//Det6:=a11*a22*a33*a44*a55*a66 - a11*a22*a33*a44*a56*a65 - a11*a22*a33*a45*a54*a66 + a11*a22*a33*a45*a56*a64 + a11*a22*a33*a46*a54*a65 - a11*a22*a33*a46*a55*a64 - a11*a22*a34*a43*a55*a66 + a11*a22*a34*a43*a56*a65 + a11*a22*a34*a45*a53*a66 - a11*a22*a34*a45*a56*a63 - a11*a22*a34*a46*a53*a65 + a11*a22*a34*a46*a55*a63 + a11*a22*a35*a43*a54*a66 - a11*a22*a35*a43*a56*a64 - a11*a22*a35*a44*a53*a66 + a11*a22*a35*a44*a56*a63 + a11*a22*a35*a46*a53*a64 - a11*a22*a35*a46*a54*a63 - a11*a22*a36*a43*a54*a65 + a11*a22*a36*a43*a55*a64 + a11*a22*a36*a44*a53*a65 - a11*a22*a36*a44*a55*a63 - a11*a22*a36*a45*a53*a64 + a11*a22*a36*a45*a54*a63 - a11*a23*a32*a44*a55*a66 + a11*a23*a32*a44*a56*a65 + a11*a23*a32*a45*a54*a66 - a11*a23*a32*a45*a56*a64 - a11*a23*a32*a46*a54*a65 + a11*a23*a32*a46*a55*a64 + a11*a23*a34*a42*a55*a66 - a11*a23*a34*a42*a56*a65 - a11*a23*a34*a45*a52*a66 + a11*a23*a34*a45*a56*a62 + a11*a23*a34*a46*a52*a65 - a11*a23*a34*a46*a55*a62 - a11*a23*a35*a42*a54*a66 + a11*a23*a35*a42*a56*a64 + a11*a23*a35*a44*a52*a66 - a11*a23*a35*a44*a56*a62 - a11*a23*a35*a46*a52*a64 + a11*a23*a35*a46*a54*a62 + a11*a23*a36*a42*a54*a65 - a11*a23*a36*a42*a55*a64 - a11*a23*a36*a44*a52*a65 + a11*a23*a36*a44*a55*a62 + a11*a23*a36*a45*a52*a64 - a11*a23*a36*a45*a54*a62 + a11*a24*a32*a43*a55*a66 - a11*a24*a32*a43*a56*a65 - a11*a24*a32*a45*a53*a66 + a11*a24*a32*a45*a56*a63 + a11*a24*a32*a46*a53*a65 - a11*a24*a32*a46*a55*a63 - a11*a24*a33*a42*a55*a66 + a11*a24*a33*a42*a56*a65 + a11*a24*a33*a45*a52*a66 - a11*a24*a33*a45*a56*a62 - a11*a24*a33*a46*a52*a65 + a11*a24*a33*a46*a55*a62 + a11*a24*a35*a42*a53*a66 - a11*a24*a35*a42*a56*a63 - a11*a24*a35*a43*a52*a66 + a11*a24*a35*a43*a56*a62 + a11*a24*a35*a46*a52*a63 - a11*a24*a35*a46*a53*a62 - a11*a24*a36*a42*a53*a65 + a11*a24*a36*a42*a55*a63 + a11*a24*a36*a43*a52*a65 - a11*a24*a36*a43*a55*a62 - a11*a24*a36*a45*a52*a63 + a11*a24*a36*a45*a53*a62 - a11*a25*a32*a43*a54*a66 + a11*a25*a32*a43*a56*a64 + a11*a25*a32*a44*a53*a66 - a11*a25*a32*a44*a56*a63 - a11*a25*a32*a46*a53*a64 + a11*a25*a32*a46*a54*a63 + a11*a25*a33*a42*a54*a66 - a11*a25*a33*a42*a56*a64 - a11*a25*a33*a44*a52*a66 + a11*a25*a33*a44*a56*a62 + a11*a25*a33*a46*a52*a64 - a11*a25*a33*a46*a54*a62 - a11*a25*a34*a42*a53*a66 + a11*a25*a34*a42*a56*a63 + a11*a25*a34*a43*a52*a66 - a11*a25*a34*a43*a56*a62 - a11*a25*a34*a46*a52*a63 + a11*a25*a34*a46*a53*a62 + a11*a25*a36*a42*a53*a64 - a11*a25*a36*a42*a54*a63 - a11*a25*a36*a43*a52*a64 + a11*a25*a36*a43*a54*a62 + a11*a25*a36*a44*a52*a63 - a11*a25*a36*a44*a53*a62 + a11*a26*a32*a43*a54*a65 - a11*a26*a32*a43*a55*a64 - a11*a26*a32*a44*a53*a65 + a11*a26*a32*a44*a55*a63 + a11*a26*a32*a45*a53*a64 - a11*a26*a32*a45*a54*a63 - a11*a26*a33*a42*a54*a65 + a11*a26*a33*a42*a55*a64 + a11*a26*a33*a44*a52*a65 - a11*a26*a33*a44*a55*a62 - a11*a26*a33*a45*a52*a64 + a11*a26*a33*a45*a54*a62 + a11*a26*a34*a42*a53*a65 - a11*a26*a34*a42*a55*a63 - a11*a26*a34*a43*a52*a65 + a11*a26*a34*a43*a55*a62 + a11*a26*a34*a45*a52*a63 - a11*a26*a34*a45*a53*a62 - a11*a26*a35*a42*a53*a64 + a11*a26*a35*a42*a54*a63 + a11*a26*a35*a43*a52*a64 - a11*a26*a35*a43*a54*a62 - a11*a26*a35*a44*a52*a63 + a11*a26*a35*a44*a53*a62 - a12*a21*a33*a44*a55*a66 + a12*a21*a33*a44*a56*a65 + a12*a21*a33*a45*a54*a66 - a12*a21*a33*a45*a56*a64 - a12*a21*a33*a46*a54*a65 + a12*a21*a33*a46*a55*a64 + a12*a21*a34*a43*a55*a66 - a12*a21*a34*a43*a56*a65 - a12*a21*a34*a45*a53*a66 + a12*a21*a34*a45*a56*a63 + a12*a21*a34*a46*a53*a65 - a12*a21*a34*a46*a55*a63 - a12*a21*a35*a43*a54*a66 + a12*a21*a35*a43*a56*a64 + a12*a21*a35*a44*a53*a66 - a12*a21*a35*a44*a56*a63 - a12*a21*a35*a46*a53*a64 + a12*a21*a35*a46*a54*a63 + a12*a21*a36*a43*a54*a65 - a12*a21*a36*a43*a55*a64 - a12*a21*a36*a44*a53*a65 + a12*a21*a36*a44*a55*a63 + a12*a21*a36*a45*a53*a64 - a12*a21*a36*a45*a54*a63 + a12*a23*a31*a44*a55*a66 - a12*a23*a31*a44*a56*a65 - a12*a23*a31*a45*a54*a66 + a12*a23*a31*a45*a56*a64 + a12*a23*a31*a46*a54*a65 - a12*a23*a31*a46*a55*a64 - a12*a23*a34*a41*a55*a66 + a12*a23*a34*a41*a56*a65 + a12*a23*a34*a45*a51*a66 - a12*a23*a34*a45*a56*a61 - a12*a23*a34*a46*a51*a65 + a12*a23*a34*a46*a55*a61 + a12*a23*a35*a41*a54*a66 - a12*a23*a35*a41*a56*a64 - a12*a23*a35*a44*a51*a66 + a12*a23*a35*a44*a56*a61 + a12*a23*a35*a46*a51*a64 - a12*a23*a35*a46*a54*a61 - a12*a23*a36*a41*a54*a65 + a12*a23*a36*a41*a55*a64 + a12*a23*a36*a44*a51*a65 - a12*a23*a36*a44*a55*a61 - a12*a23*a36*a45*a51*a64 + a12*a23*a36*a45*a54*a61 - a12*a24*a31*a43*a55*a66 + a12*a24*a31*a43*a56*a65 + a12*a24*a31*a45*a53*a66 - a12*a24*a31*a45*a56*a63 - a12*a24*a31*a46*a53*a65 + a12*a24*a31*a46*a55*a63 + a12*a24*a33*a41*a55*a66 - a12*a24*a33*a41*a56*a65 - a12*a24*a33*a45*a51*a66 + a12*a24*a33*a45*a56*a61 + a12*a24*a33*a46*a51*a65 - a12*a24*a33*a46*a55*a61 - a12*a24*a35*a41*a53*a66 + a12*a24*a35*a41*a56*a63 + a12*a24*a35*a43*a51*a66 - a12*a24*a35*a43*a56*a61 - a12*a24*a35*a46*a51*a63 + a12*a24*a35*a46*a53*a61 + a12*a24*a36*a41*a53*a65 - a12*a24*a36*a41*a55*a63 - a12*a24*a36*a43*a51*a65 + a12*a24*a36*a43*a55*a61 + a12*a24*a36*a45*a51*a63 - a12*a24*a36*a45*a53*a61 + a12*a25*a31*a43*a54*a66 - a12*a25*a31*a43*a56*a64 - a12*a25*a31*a44*a53*a66 + a12*a25*a31*a44*a56*a63 + a12*a25*a31*a46*a53*a64 - a12*a25*a31*a46*a54*a63 - a12*a25*a33*a41*a54*a66 + a12*a25*a33*a41*a56*a64 + a12*a25*a33*a44*a51*a66 - a12*a25*a33*a44*a56*a61 - a12*a25*a33*a46*a51*a64 + a12*a25*a33*a46*a54*a61 + a12*a25*a34*a41*a53*a66 - a12*a25*a34*a41*a56*a63 - a12*a25*a34*a43*a51*a66 + a12*a25*a34*a43*a56*a61 + a12*a25*a34*a46*a51*a63 - a12*a25*a34*a46*a53*a61 - a12*a25*a36*a41*a53*a64 + a12*a25*a36*a41*a54*a63 + a12*a25*a36*a43*a51*a64 - a12*a25*a36*a43*a54*a61 - a12*a25*a36*a44*a51*a63 + a12*a25*a36*a44*a53*a61 - a12*a26*a31*a43*a54*a65 + a12*a26*a31*a43*a55*a64 + a12*a26*a31*a44*a53*a65 - a12*a26*a31*a44*a55*a63 - a12*a26*a31*a45*a53*a64 + a12*a26*a31*a45*a54*a63 + a12*a26*a33*a41*a54*a65 - a12*a26*a33*a41*a55*a64 - a12*a26*a33*a44*a51*a65 + a12*a26*a33*a44*a55*a61 + a12*a26*a33*a45*a51*a64 - a12*a26*a33*a45*a54*a61 - a12*a26*a34*a41*a53*a65 + a12*a26*a34*a41*a55*a63 + a12*a26*a34*a43*a51*a65 - a12*a26*a34*a43*a55*a61 - a12*a26*a34*a45*a51*a63 + a12*a26*a34*a45*a53*a61 + a12*a26*a35*a41*a53*a64 - a12*a26*a35*a41*a54*a63 - a12*a26*a35*a43*a51*a64 + a12*a26*a35*a43*a54*a61 + a12*a26*a35*a44*a51*a63 - a12*a26*a35*a44*a53*a61 + a13*a21*a32*a44*a55*a66 - a13*a21*a32*a44*a56*a65 - a13*a21*a32*a45*a54*a66 + a13*a21*a32*a45*a56*a64 + a13*a21*a32*a46*a54*a65 - a13*a21*a32*a46*a55*a64 - a13*a21*a34*a42*a55*a66 + a13*a21*a34*a42*a56*a65 + a13*a21*a34*a45*a52*a66 - a13*a21*a34*a45*a56*a62 - a13*a21*a34*a46*a52*a65 + a13*a21*a34*a46*a55*a62 + a13*a21*a35*a42*a54*a66 - a13*a21*a35*a42*a56*a64 - a13*a21*a35*a44*a52*a66 + a13*a21*a35*a44*a56*a62 + a13*a21*a35*a46*a52*a64 - a13*a21*a35*a46*a54*a62 - a13*a21*a36*a42*a54*a65 + a13*a21*a36*a42*a55*a64 + a13*a21*a36*a44*a52*a65 - a13*a21*a36*a44*a55*a62 - a13*a21*a36*a45*a52*a64 + a13*a21*a36*a45*a54*a62 - a13*a22*a31*a44*a55*a66 + a13*a22*a31*a44*a56*a65 + a13*a22*a31*a45*a54*a66 - a13*a22*a31*a45*a56*a64 - a13*a22*a31*a46*a54*a65 + a13*a22*a31*a46*a55*a64 + a13*a22*a34*a41*a55*a66 - a13*a22*a34*a41*a56*a65 - a13*a22*a34*a45*a51*a66 + a13*a22*a34*a45*a56*a61 + a13*a22*a34*a46*a51*a65 - a13*a22*a34*a46*a55*a61 - a13*a22*a35*a41*a54*a66 + a13*a22*a35*a41*a56*a64 + a13*a22*a35*a44*a51*a66 - a13*a22*a35*a44*a56*a61 - a13*a22*a35*a46*a51*a64 + a13*a22*a35*a46*a54*a61 + a13*a22*a36*a41*a54*a65 - a13*a22*a36*a41*a55*a64 - a13*a22*a36*a44*a51*a65 + a13*a22*a36*a44*a55*a61 + a13*a22*a36*a45*a51*a64 - a13*a22*a36*a45*a54*a61 + a13*a24*a31*a42*a55*a66 - a13*a24*a31*a42*a56*a65 - a13*a24*a31*a45*a52*a66 + a13*a24*a31*a45*a56*a62 + a13*a24*a31*a46*a52*a65 - a13*a24*a31*a46*a55*a62 - a13*a24*a32*a41*a55*a66 + a13*a24*a32*a41*a56*a65 + a13*a24*a32*a45*a51*a66 - a13*a24*a32*a45*a56*a61 - a13*a24*a32*a46*a51*a65 + a13*a24*a32*a46*a55*a61 + a13*a24*a35*a41*a52*a66 - a13*a24*a35*a41*a56*a62 - a13*a24*a35*a42*a51*a66 + a13*a24*a35*a42*a56*a61 + a13*a24*a35*a46*a51*a62 - a13*a24*a35*a46*a52*a61 - a13*a24*a36*a41*a52*a65 + a13*a24*a36*a41*a55*a62 + a13*a24*a36*a42*a51*a65 - a13*a24*a36*a42*a55*a61 - a13*a24*a36*a45*a51*a62 + a13*a24*a36*a45*a52*a61 - a13*a25*a31*a42*a54*a66 + a13*a25*a31*a42*a56*a64 + a13*a25*a31*a44*a52*a66 - a13*a25*a31*a44*a56*a62 - a13*a25*a31*a46*a52*a64 + a13*a25*a31*a46*a54*a62 + a13*a25*a32*a41*a54*a66 - a13*a25*a32*a41*a56*a64 - a13*a25*a32*a44*a51*a66 + a13*a25*a32*a44*a56*a61 + a13*a25*a32*a46*a51*a64 - a13*a25*a32*a46*a54*a61 - a13*a25*a34*a41*a52*a66 + a13*a25*a34*a41*a56*a62 + a13*a25*a34*a42*a51*a66 - a13*a25*a34*a42*a56*a61 - a13*a25*a34*a46*a51*a62 + a13*a25*a34*a46*a52*a61 + a13*a25*a36*a41*a52*a64 - a13*a25*a36*a41*a54*a62 - a13*a25*a36*a42*a51*a64 + a13*a25*a36*a42*a54*a61 + a13*a25*a36*a44*a51*a62 - a13*a25*a36*a44*a52*a61 + a13*a26*a31*a42*a54*a65 - a13*a26*a31*a42*a55*a64 - a13*a26*a31*a44*a52*a65 + a13*a26*a31*a44*a55*a62 + a13*a26*a31*a45*a52*a64 - a13*a26*a31*a45*a54*a62 - a13*a26*a32*a41*a54*a65 + a13*a26*a32*a41*a55*a64 + a13*a26*a32*a44*a51*a65 - a13*a26*a32*a44*a55*a61 - a13*a26*a32*a45*a51*a64 + a13*a26*a32*a45*a54*a61 + a13*a26*a34*a41*a52*a65 - a13*a26*a34*a41*a55*a62 - a13*a26*a34*a42*a51*a65 + a13*a26*a34*a42*a55*a61 + a13*a26*a34*a45*a51*a62 - a13*a26*a34*a45*a52*a61 - a13*a26*a35*a41*a52*a64 + a13*a26*a35*a41*a54*a62 + a13*a26*a35*a42*a51*a64 - a13*a26*a35*a42*a54*a61 - a13*a26*a35*a44*a51*a62 + a13*a26*a35*a44*a52*a61 - a14*a21*a32*a43*a55*a66 + a14*a21*a32*a43*a56*a65 + a14*a21*a32*a45*a53*a66 - a14*a21*a32*a45*a56*a63 - a14*a21*a32*a46*a53*a65 + a14*a21*a32*a46*a55*a63 + a14*a21*a33*a42*a55*a66 - a14*a21*a33*a42*a56*a65 - a14*a21*a33*a45*a52*a66 + a14*a21*a33*a45*a56*a62 + a14*a21*a33*a46*a52*a65 - a14*a21*a33*a46*a55*a62 - a14*a21*a35*a42*a53*a66 + a14*a21*a35*a42*a56*a63 + a14*a21*a35*a43*a52*a66 - a14*a21*a35*a43*a56*a62 - a14*a21*a35*a46*a52*a63 + a14*a21*a35*a46*a53*a62 + a14*a21*a36*a42*a53*a65 - a14*a21*a36*a42*a55*a63 - a14*a21*a36*a43*a52*a65 + a14*a21*a36*a43*a55*a62 + a14*a21*a36*a45*a52*a63 - a14*a21*a36*a45*a53*a62 + a14*a22*a31*a43*a55*a66 - a14*a22*a31*a43*a56*a65 - a14*a22*a31*a45*a53*a66 + a14*a22*a31*a45*a56*a63 + a14*a22*a31*a46*a53*a65 - a14*a22*a31*a46*a55*a63 - a14*a22*a33*a41*a55*a66 + a14*a22*a33*a41*a56*a65 + a14*a22*a33*a45*a51*a66 - a14*a22*a33*a45*a56*a61 - a14*a22*a33*a46*a51*a65 + a14*a22*a33*a46*a55*a61 + a14*a22*a35*a41*a53*a66 - a14*a22*a35*a41*a56*a63 - a14*a22*a35*a43*a51*a66 + a14*a22*a35*a43*a56*a61 + a14*a22*a35*a46*a51*a63 - a14*a22*a35*a46*a53*a61 - a14*a22*a36*a41*a53*a65 + a14*a22*a36*a41*a55*a63 + a14*a22*a36*a43*a51*a65 - a14*a22*a36*a43*a55*a61 - a14*a22*a36*a45*a51*a63 + a14*a22*a36*a45*a53*a61 - a14*a23*a31*a42*a55*a66 + a14*a23*a31*a42*a56*a65 + a14*a23*a31*a45*a52*a66 - a14*a23*a31*a45*a56*a62 - a14*a23*a31*a46*a52*a65 + a14*a23*a31*a46*a55*a62 + a14*a23*a32*a41*a55*a66 - a14*a23*a32*a41*a56*a65 - a14*a23*a32*a45*a51*a66 + a14*a23*a32*a45*a56*a61 + a14*a23*a32*a46*a51*a65 - a14*a23*a32*a46*a55*a61 - a14*a23*a35*a41*a52*a66 + a14*a23*a35*a41*a56*a62 + a14*a23*a35*a42*a51*a66 - a14*a23*a35*a42*a56*a61 - a14*a23*a35*a46*a51*a62 + a14*a23*a35*a46*a52*a61 + a14*a23*a36*a41*a52*a65 - a14*a23*a36*a41*a55*a62 - a14*a23*a36*a42*a51*a65 + a14*a23*a36*a42*a55*a61 + a14*a23*a36*a45*a51*a62 - a14*a23*a36*a45*a52*a61 + a14*a25*a31*a42*a53*a66 - a14*a25*a31*a42*a56*a63 - a14*a25*a31*a43*a52*a66 + a14*a25*a31*a43*a56*a62 + a14*a25*a31*a46*a52*a63 - a14*a25*a31*a46*a53*a62 - a14*a25*a32*a41*a53*a66 + a14*a25*a32*a41*a56*a63 + a14*a25*a32*a43*a51*a66 - a14*a25*a32*a43*a56*a61 - a14*a25*a32*a46*a51*a63 + a14*a25*a32*a46*a53*a61 + a14*a25*a33*a41*a52*a66 - a14*a25*a33*a41*a56*a62 - a14*a25*a33*a42*a51*a66 + a14*a25*a33*a42*a56*a61 + a14*a25*a33*a46*a51*a62 - a14*a25*a33*a46*a52*a61 - a14*a25*a36*a41*a52*a63 + a14*a25*a36*a41*a53*a62 + a14*a25*a36*a42*a51*a63 - a14*a25*a36*a42*a53*a61 - a14*a25*a36*a43*a51*a62 + a14*a25*a36*a43*a52*a61 - a14*a26*a31*a42*a53*a65 + a14*a26*a31*a42*a55*a63 + a14*a26*a31*a43*a52*a65 - a14*a26*a31*a43*a55*a62 - a14*a26*a31*a45*a52*a63 + a14*a26*a31*a45*a53*a62 + a14*a26*a32*a41*a53*a65 - a14*a26*a32*a41*a55*a63 - a14*a26*a32*a43*a51*a65 + a14*a26*a32*a43*a55*a61 + a14*a26*a32*a45*a51*a63 - a14*a26*a32*a45*a53*a61 - a14*a26*a33*a41*a52*a65 + a14*a26*a33*a41*a55*a62 + a14*a26*a33*a42*a51*a65 - a14*a26*a33*a42*a55*a61 - a14*a26*a33*a45*a51*a62 + a14*a26*a33*a45*a52*a61 + a14*a26*a35*a41*a52*a63 - a14*a26*a35*a41*a53*a62 - a14*a26*a35*a42*a51*a63 + a14*a26*a35*a42*a53*a61 + a14*a26*a35*a43*a51*a62 - a14*a26*a35*a43*a52*a61 + a15*a21*a32*a43*a54*a66 - a15*a21*a32*a43*a56*a64 - a15*a21*a32*a44*a53*a66 + a15*a21*a32*a44*a56*a63 + a15*a21*a32*a46*a53*a64 - a15*a21*a32*a46*a54*a63 - a15*a21*a33*a42*a54*a66 + a15*a21*a33*a42*a56*a64 + a15*a21*a33*a44*a52*a66 - a15*a21*a33*a44*a56*a62 - a15*a21*a33*a46*a52*a64 + a15*a21*a33*a46*a54*a62 + a15*a21*a34*a42*a53*a66 - a15*a21*a34*a42*a56*a63 - a15*a21*a34*a43*a52*a66 + a15*a21*a34*a43*a56*a62 + a15*a21*a34*a46*a52*a63 - a15*a21*a34*a46*a53*a62 - a15*a21*a36*a42*a53*a64 + a15*a21*a36*a42*a54*a63 + a15*a21*a36*a43*a52*a64 - a15*a21*a36*a43*a54*a62 - a15*a21*a36*a44*a52*a63 + a15*a21*a36*a44*a53*a62 - a15*a22*a31*a43*a54*a66 + a15*a22*a31*a43*a56*a64 + a15*a22*a31*a44*a53*a66 - a15*a22*a31*a44*a56*a63 - a15*a22*a31*a46*a53*a64 + a15*a22*a31*a46*a54*a63 + a15*a22*a33*a41*a54*a66 - a15*a22*a33*a41*a56*a64 - a15*a22*a33*a44*a51*a66 + a15*a22*a33*a44*a56*a61 + a15*a22*a33*a46*a51*a64 - a15*a22*a33*a46*a54*a61 - a15*a22*a34*a41*a53*a66 + a15*a22*a34*a41*a56*a63 + a15*a22*a34*a43*a51*a66 - a15*a22*a34*a43*a56*a61 - a15*a22*a34*a46*a51*a63 + a15*a22*a34*a46*a53*a61 + a15*a22*a36*a41*a53*a64 - a15*a22*a36*a41*a54*a63 - a15*a22*a36*a43*a51*a64 + a15*a22*a36*a43*a54*a61 + a15*a22*a36*a44*a51*a63 - a15*a22*a36*a44*a53*a61 + a15*a23*a31*a42*a54*a66 - a15*a23*a31*a42*a56*a64 - a15*a23*a31*a44*a52*a66 + a15*a23*a31*a44*a56*a62 + a15*a23*a31*a46*a52*a64 - a15*a23*a31*a46*a54*a62 - a15*a23*a32*a41*a54*a66 + a15*a23*a32*a41*a56*a64 + a15*a23*a32*a44*a51*a66 - a15*a23*a32*a44*a56*a61 - a15*a23*a32*a46*a51*a64 + a15*a23*a32*a46*a54*a61 + a15*a23*a34*a41*a52*a66 - a15*a23*a34*a41*a56*a62 - a15*a23*a34*a42*a51*a66 + a15*a23*a34*a42*a56*a61 + a15*a23*a34*a46*a51*a62 - a15*a23*a34*a46*a52*a61 - a15*a23*a36*a41*a52*a64 + a15*a23*a36*a41*a54*a62 + a15*a23*a36*a42*a51*a64 - a15*a23*a36*a42*a54*a61 - a15*a23*a36*a44*a51*a62 + a15*a23*a36*a44*a52*a61 - a15*a24*a31*a42*a53*a66 + a15*a24*a31*a42*a56*a63 + a15*a24*a31*a43*a52*a66 - a15*a24*a31*a43*a56*a62 - a15*a24*a31*a46*a52*a63 + a15*a24*a31*a46*a53*a62 + a15*a24*a32*a41*a53*a66 - a15*a24*a32*a41*a56*a63 - a15*a24*a32*a43*a51*a66 + a15*a24*a32*a43*a56*a61 + a15*a24*a32*a46*a51*a63 - a15*a24*a32*a46*a53*a61 - a15*a24*a33*a41*a52*a66 + a15*a24*a33*a41*a56*a62 + a15*a24*a33*a42*a51*a66 - a15*a24*a33*a42*a56*a61 - a15*a24*a33*a46*a51*a62 + a15*a24*a33*a46*a52*a61 + a15*a24*a36*a41*a52*a63 - a15*a24*a36*a41*a53*a62 - a15*a24*a36*a42*a51*a63 + a15*a24*a36*a42*a53*a61 + a15*a24*a36*a43*a51*a62 - a15*a24*a36*a43*a52*a61 + a15*a26*a31*a42*a53*a64 - a15*a26*a31*a42*a54*a63 - a15*a26*a31*a43*a52*a64 + a15*a26*a31*a43*a54*a62 + a15*a26*a31*a44*a52*a63 - a15*a26*a31*a44*a53*a62 - a15*a26*a32*a41*a53*a64 + a15*a26*a32*a41*a54*a63 + a15*a26*a32*a43*a51*a64 - a15*a26*a32*a43*a54*a61 - a15*a26*a32*a44*a51*a63 + a15*a26*a32*a44*a53*a61 + a15*a26*a33*a41*a52*a64 - a15*a26*a33*a41*a54*a62 - a15*a26*a33*a42*a51*a64 + a15*a26*a33*a42*a54*a61 + a15*a26*a33*a44*a51*a62 - a15*a26*a33*a44*a52*a61 - a15*a26*a34*a41*a52*a63 + a15*a26*a34*a41*a53*a62 + a15*a26*a34*a42*a51*a63 - a15*a26*a34*a42*a53*a61 - a15*a26*a34*a43*a51*a62 + a15*a26*a34*a43*a52*a61 - a16*a21*a32*a43*a54*a65 + a16*a21*a32*a43*a55*a64 + a16*a21*a32*a44*a53*a65 - a16*a21*a32*a44*a55*a63 - a16*a21*a32*a45*a53*a64 + a16*a21*a32*a45*a54*a63 + a16*a21*a33*a42*a54*a65 - a16*a21*a33*a42*a55*a64 - a16*a21*a33*a44*a52*a65 + a16*a21*a33*a44*a55*a62 + a16*a21*a33*a45*a52*a64 - a16*a21*a33*a45*a54*a62 - a16*a21*a34*a42*a53*a65 + a16*a21*a34*a42*a55*a63 + a16*a21*a34*a43*a52*a65 - a16*a21*a34*a43*a55*a62 - a16*a21*a34*a45*a52*a63 + a16*a21*a34*a45*a53*a62 + a16*a21*a35*a42*a53*a64 - a16*a21*a35*a42*a54*a63 - a16*a21*a35*a43*a52*a64 + a16*a21*a35*a43*a54*a62 + a16*a21*a35*a44*a52*a63 - a16*a21*a35*a44*a53*a62 + a16*a22*a31*a43*a54*a65 - a16*a22*a31*a43*a55*a64 - a16*a22*a31*a44*a53*a65 + a16*a22*a31*a44*a55*a63 + a16*a22*a31*a45*a53*a64 - a16*a22*a31*a45*a54*a63 - a16*a22*a33*a41*a54*a65 + a16*a22*a33*a41*a55*a64 + a16*a22*a33*a44*a51*a65 - a16*a22*a33*a44*a55*a61 - a16*a22*a33*a45*a51*a64 + a16*a22*a33*a45*a54*a61 + a16*a22*a34*a41*a53*a65 - a16*a22*a34*a41*a55*a63 - a16*a22*a34*a43*a51*a65 + a16*a22*a34*a43*a55*a61 + a16*a22*a34*a45*a51*a63 - a16*a22*a34*a45*a53*a61 - a16*a22*a35*a41*a53*a64 + a16*a22*a35*a41*a54*a63 + a16*a22*a35*a43*a51*a64 - a16*a22*a35*a43*a54*a61 - a16*a22*a35*a44*a51*a63 + a16*a22*a35*a44*a53*a61 - a16*a23*a31*a42*a54*a65 + a16*a23*a31*a42*a55*a64 + a16*a23*a31*a44*a52*a65 - a16*a23*a31*a44*a55*a62 - a16*a23*a31*a45*a52*a64 + a16*a23*a31*a45*a54*a62 + a16*a23*a32*a41*a54*a65 - a16*a23*a32*a41*a55*a64 - a16*a23*a32*a44*a51*a65 + a16*a23*a32*a44*a55*a61 + a16*a23*a32*a45*a51*a64 - a16*a23*a32*a45*a54*a61 - a16*a23*a34*a41*a52*a65 + a16*a23*a34*a41*a55*a62 + a16*a23*a34*a42*a51*a65 - a16*a23*a34*a42*a55*a61 - a16*a23*a34*a45*a51*a62 + a16*a23*a34*a45*a52*a61 + a16*a23*a35*a41*a52*a64 - a16*a23*a35*a41*a54*a62 - a16*a23*a35*a42*a51*a64 + a16*a23*a35*a42*a54*a61 + a16*a23*a35*a44*a51*a62 - a16*a23*a35*a44*a52*a61 + a16*a24*a31*a42*a53*a65 - a16*a24*a31*a42*a55*a63 - a16*a24*a31*a43*a52*a65 + a16*a24*a31*a43*a55*a62 + a16*a24*a31*a45*a52*a63 - a16*a24*a31*a45*a53*a62 - a16*a24*a32*a41*a53*a65 + a16*a24*a32*a41*a55*a63 + a16*a24*a32*a43*a51*a65 - a16*a24*a32*a43*a55*a61 - a16*a24*a32*a45*a51*a63 + a16*a24*a32*a45*a53*a61 + a16*a24*a33*a41*a52*a65 - a16*a24*a33*a41*a55*a62 - a16*a24*a33*a42*a51*a65 + a16*a24*a33*a42*a55*a61 + a16*a24*a33*a45*a51*a62 - a16*a24*a33*a45*a52*a61 - a16*a24*a35*a41*a52*a63 + a16*a24*a35*a41*a53*a62 + a16*a24*a35*a42*a51*a63 - a16*a24*a35*a42*a53*a61 - a16*a24*a35*a43*a51*a62 + a16*a24*a35*a43*a52*a61 - a16*a25*a31*a42*a53*a64 + a16*a25*a31*a42*a54*a63 + a16*a25*a31*a43*a52*a64 - a16*a25*a31*a43*a54*a62 - a16*a25*a31*a44*a52*a63 + a16*a25*a31*a44*a53*a62 + a16*a25*a32*a41*a53*a64 - a16*a25*a32*a41*a54*a63 - a16*a25*a32*a43*a51*a64 + a16*a25*a32*a43*a54*a61 + a16*a25*a32*a44*a51*a63 - a16*a25*a32*a44*a53*a61 - a16*a25*a33*a41*a52*a64 + a16*a25*a33*a41*a54*a62 + a16*a25*a33*a42*a51*a64 - a16*a25*a33*a42*a54*a61 - a16*a25*a33*a44*a51*a62 + a16*a25*a33*a44*a52*a61 + a16*a25*a34*a41*a52*a63 - a16*a25*a34*a41*a53*a62 - a16*a25*a34*a42*a51*a63 + a16*a25*a34*a42*a53*a61 + a16*a25*a34*a43*a51*a62 - a16*a25*a34*a43*a52*a61;
Det6:=((a31*a42*a54*a63 - a31*a42*a53*a64 + a31*a43*a52*a64 - a31*a43*a54*a62 - a31*a44*a52*a63 + a31*a44*a53*a62 + a32*a41*a53*a64 - a32*a41*a54*a63 - a32*a43*a51*a64 + a32*a43*a54*a61 + a32*a44*a51*a63 - a32*a44*a53*a61 - a33*a41*a52*a64 + a33*a41*a54*a62 + a33*a42*a51*a64 - a33*a42*a54*a61 - a33*a44*a51*a62 + a33*a44*a52*a61 + a34*a41*a52*a63 - a34*a41*a53*a62 - a34*a42*a51*a63 + a34*a42*a53*a61 + a34*a43*a51*a62 - a34*a43*a52*a61)*a25 + (a31*a42*a53*a65 - a31*a42*a55*a63 - a31*a43*a52*a65 + a31*a43*a55*a62 + a31*a45*a52*a63 - a31*a45*a53*a62 - a32*a41*a53*a65 + a32*a41*a55*a63 + a32*a43*a51*a65 - a32*a43*a55*a61 - a32*a45*a51*a63 + a32*a45*a53*a61 + a33*a41*a52*a65 - a33*a41*a55*a62 - a33*a42*a51*a65 + a33*a42*a55*a61 + a33*a45*a51*a62 - a33*a45*a52*a61 - a35*a41*a52*a63 + a35*a41*a53*a62 + a35*a42*a51*a63 - a35*a42*a53*a61 - a35*a43*a51*a62 + a35*a43*a52*a61)*a24 + (a31*a42*a55*a64 - a31*a42*a54*a65 + a31*a44*a52*a65 - a31*a44*a55*a62 - a31*a45*a52*a64 + a31*a45*a54*a62 + a32*a41*a54*a65 - a32*a41*a55*a64 - a32*a44*a51*a65 + a32*a44*a55*a61 + a32*a45*a51*a64 - a32*a45*a54*a61 - a34*a41*a52*a65 + a34*a41*a55*a62 + a34*a42*a51*a65 - a34*a42*a55*a61 - a34*a45*a51*a62 + a34*a45*a52*a61 + a35*a41*a52*a64 - a35*a41*a54*a62 - a35*a42*a51*a64 + a35*a42*a54*a61 + a35*a44*a51*a62 - a35*a44*a52*a61)*a23 + (a31*a43*a54*a65 - a31*a43*a55*a64 - a31*a44*a53*a65 + a31*a44*a55*a63 + a31*a45*a53*a64 - a31*a45*a54*a63 - a33*a41*a54*a65 + a33*a41*a55*a64 + a33*a44*a51*a65 - a33*a44*a55*a61 - a33*a45*a51*a64 + a33*a45*a54*a61 + a34*a41*a53*a65 - a34*a41*a55*a63 - a34*a43*a51*a65 + a34*a43*a55*a61 + a34*a45*a51*a63 - a34*a45*a53*a61 - a35*a41*a53*a64 + a35*a41*a54*a63 + a35*a43*a51*a64 - a35*a43*a54*a61 - a35*a44*a51*a63 + a35*a44*a53*a61)*a22 + (a32*a43*a55*a64 - a32*a43*a54*a65 + a32*a44*a53*a65 - a32*a44*a55*a63 - a32*a45*a53*a64 + a32*a45*a54*a63 + a33*a42*a54*a65 - a33*a42*a55*a64 - a33*a44*a52*a65 + a33*a44*a55*a62 + a33*a45*a52*a64 - a33*a45*a54*a62 - a34*a42*a53*a65 + a34*a42*a55*a63 + a34*a43*a52*a65 - a34*a43*a55*a62 - a34*a45*a52*a63 + a34*a45*a53*a62 + a35*a42*a53*a64 - a35*a42*a54*a63 - a35*a43*a52*a64 + a35*a43*a54*a62 + a35*a44*a52*a63 - a35*a44*a53*a62)*a21)*a16 
	+ ((a31*a42*a53*a64 - a31*a42*a54*a63 - a31*a43*a52*a64 + a31*a43*a54*a62 + a31*a44*a52*a63 - a31*a44*a53*a62 - a32*a41*a53*a64 + a32*a41*a54*a63 + a32*a43*a51*a64 - a32*a43*a54*a61 - a32*a44*a51*a63 + a32*a44*a53*a61 + a33*a41*a52*a64 - a33*a41*a54*a62 - a33*a42*a51*a64 + a33*a42*a54*a61 + a33*a44*a51*a62 - a33*a44*a52*a61 - a34*a41*a52*a63 + a34*a41*a53*a62 + a34*a42*a51*a63 - a34*a42*a53*a61 - a34*a43*a51*a62 + a34*a43*a52*a61)*a26 + (a31*a42*a56*a63 - a31*a42*a53*a66 + a31*a43*a52*a66 - a31*a43*a56*a62 - a31*a46*a52*a63 + a31*a46*a53*a62 + a32*a41*a53*a66 - a32*a41*a56*a63 - a32*a43*a51*a66 + a32*a43*a56*a61 + a32*a46*a51*a63 - a32*a46*a53*a61 - a33*a41*a52*a66 + a33*a41*a56*a62 + a33*a42*a51*a66 - a33*a42*a56*a61 - a33*a46*a51*a62 + a33*a46*a52*a61 + a36*a41*a52*a63 - a36*a41*a53*a62 - a36*a42*a51*a63 + a36*a42*a53*a61 + a36*a43*a51*a62 - a36*a43*a52*a61)*a24 + (a31*a42*a54*a66 - a31*a42*a56*a64 - a31*a44*a52*a66 + a31*a44*a56*a62 + a31*a46*a52*a64 - a31*a46*a54*a62 - a32*a41*a54*a66 + a32*a41*a56*a64 + a32*a44*a51*a66 - a32*a44*a56*a61 - a32*a46*a51*a64 + a32*a46*a54*a61 + a34*a41*a52*a66 - a34*a41*a56*a62 - a34*a42*a51*a66 + a34*a42*a56*a61 + a34*a46*a51*a62 - a34*a46*a52*a61 - a36*a41*a52*a64 + a36*a41*a54*a62 + a36*a42*a51*a64 - a36*a42*a54*a61 - a36*a44*a51*a62 + a36*a44*a52*a61)*a23 + (a31*a43*a56*a64 - a31*a43*a54*a66 + a31*a44*a53*a66 - a31*a44*a56*a63 - a31*a46*a53*a64 + a31*a46*a54*a63 + a33*a41*a54*a66 - a33*a41*a56*a64 - a33*a44*a51*a66 + a33*a44*a56*a61 + a33*a46*a51*a64 - a33*a46*a54*a61 - a34*a41*a53*a66 + a34*a41*a56*a63 + a34*a43*a51*a66 - a34*a43*a56*a61 - a34*a46*a51*a63 + a34*a46*a53*a61 + a36*a41*a53*a64 - a36*a41*a54*a63 - a36*a43*a51*a64 + a36*a43*a54*a61 + a36*a44*a51*a63 - a36*a44*a53*a61)*a22 + (a32*a43*a54*a66 - a32*a43*a56*a64 - a32*a44*a53*a66 + a32*a44*a56*a63 + a32*a46*a53*a64 - a32*a46*a54*a63 - a33*a42*a54*a66 + a33*a42*a56*a64 + a33*a44*a52*a66 - a33*a44*a56*a62 - a33*a46*a52*a64 + a33*a46*a54*a62 + a34*a42*a53*a66 - a34*a42*a56*a63 - a34*a43*a52*a66 + a34*a43*a56*a62 + a34*a46*a52*a63 - a34*a46*a53*a62 - a36*a42*a53*a64 + a36*a42*a54*a63 + a36*a43*a52*a64 - a36*a43*a54*a62 - a36*a44*a52*a63 + a36*a44*a53*a62)*a21)*a15 
	+ ((a31*a42*a55*a63 - a31*a42*a53*a65 + a31*a43*a52*a65 - a31*a43*a55*a62 - a31*a45*a52*a63 + a31*a45*a53*a62 + a32*a41*a53*a65 - a32*a41*a55*a63 - a32*a43*a51*a65 + a32*a43*a55*a61 + a32*a45*a51*a63 - a32*a45*a53*a61 - a33*a41*a52*a65 + a33*a41*a55*a62 + a33*a42*a51*a65 - a33*a42*a55*a61 - a33*a45*a51*a62 + a33*a45*a52*a61 + a35*a41*a52*a63 - a35*a41*a53*a62 - a35*a42*a51*a63 + a35*a42*a53*a61 + a35*a43*a51*a62 - a35*a43*a52*a61)*a26 + (a31*a42*a53*a66 - a31*a42*a56*a63 - a31*a43*a52*a66 + a31*a43*a56*a62 + a31*a46*a52*a63 - a31*a46*a53*a62 - a32*a41*a53*a66 + a32*a41*a56*a63 + a32*a43*a51*a66 - a32*a43*a56*a61 - a32*a46*a51*a63 + a32*a46*a53*a61 + a33*a41*a52*a66 - a33*a41*a56*a62 - a33*a42*a51*a66 + a33*a42*a56*a61 + a33*a46*a51*a62 - a33*a46*a52*a61 - a36*a41*a52*a63 + a36*a41*a53*a62 + a36*a42*a51*a63 - a36*a42*a53*a61 - a36*a43*a51*a62 + a36*a43*a52*a61)*a25 + (a31*a42*a56*a65 - a31*a42*a55*a66 + a31*a45*a52*a66 - a31*a45*a56*a62 - a31*a46*a52*a65 + a31*a46*a55*a62 + a32*a41*a55*a66 - a32*a41*a56*a65 - a32*a45*a51*a66 + a32*a45*a56*a61 + a32*a46*a51*a65 - a32*a46*a55*a61 - a35*a41*a52*a66 + a35*a41*a56*a62 + a35*a42*a51*a66 - a35*a42*a56*a61 - a35*a46*a51*a62 + a35*a46*a52*a61 + a36*a41*a52*a65 - a36*a41*a55*a62 - a36*a42*a51*a65 + a36*a42*a55*a61 + a36*a45*a51*a62 - a36*a45*a52*a61)*a23 + (a31*a43*a55*a66 - a31*a43*a56*a65 - a31*a45*a53*a66 + a31*a45*a56*a63 + a31*a46*a53*a65 - a31*a46*a55*a63 - a33*a41*a55*a66 + a33*a41*a56*a65 + a33*a45*a51*a66 - a33*a45*a56*a61 - a33*a46*a51*a65 + a33*a46*a55*a61 + a35*a41*a53*a66 - a35*a41*a56*a63 - a35*a43*a51*a66 + a35*a43*a56*a61 + a35*a46*a51*a63 - a35*a46*a53*a61 - a36*a41*a53*a65 + a36*a41*a55*a63 + a36*a43*a51*a65 - a36*a43*a55*a61 - a36*a45*a51*a63 + a36*a45*a53*a61)*a22 + (a32*a43*a56*a65 - a32*a43*a55*a66 + a32*a45*a53*a66 - a32*a45*a56*a63 - a32*a46*a53*a65 + a32*a46*a55*a63 + a33*a42*a55*a66 - a33*a42*a56*a65 - a33*a45*a52*a66 + a33*a45*a56*a62 + a33*a46*a52*a65 - a33*a46*a55*a62 - a35*a42*a53*a66 + a35*a42*a56*a63 + a35*a43*a52*a66 - a35*a43*a56*a62 - a35*a46*a52*a63 + a35*a46*a53*a62 + a36*a42*a53*a65 - a36*a42*a55*a63 - a36*a43*a52*a65 + a36*a43*a55*a62 + a36*a45*a52*a63 - a36*a45*a53*a62)*a21)*a14 
	+ ((a31*a42*a54*a65 - a31*a42*a55*a64 - a31*a44*a52*a65 + a31*a44*a55*a62 + a31*a45*a52*a64 - a31*a45*a54*a62 - a32*a41*a54*a65 + a32*a41*a55*a64 + a32*a44*a51*a65 - a32*a44*a55*a61 - a32*a45*a51*a64 + a32*a45*a54*a61 + a34*a41*a52*a65 - a34*a41*a55*a62 - a34*a42*a51*a65 + a34*a42*a55*a61 + a34*a45*a51*a62 - a34*a45*a52*a61 - a35*a41*a52*a64 + a35*a41*a54*a62 + a35*a42*a51*a64 - a35*a42*a54*a61 - a35*a44*a51*a62 + a35*a44*a52*a61)*a26 + (a31*a42*a56*a64 - a31*a42*a54*a66 + a31*a44*a52*a66 - a31*a44*a56*a62 - a31*a46*a52*a64 + a31*a46*a54*a62 + a32*a41*a54*a66 - a32*a41*a56*a64 - a32*a44*a51*a66 + a32*a44*a56*a61 + a32*a46*a51*a64 - a32*a46*a54*a61 - a34*a41*a52*a66 + a34*a41*a56*a62 + a34*a42*a51*a66 - a34*a42*a56*a61 - a34*a46*a51*a62 + a34*a46*a52*a61 + a36*a41*a52*a64 - a36*a41*a54*a62 - a36*a42*a51*a64 + a36*a42*a54*a61 + a36*a44*a51*a62 - a36*a44*a52*a61)*a25 + (a31*a42*a55*a66 - a31*a42*a56*a65 - a31*a45*a52*a66 + a31*a45*a56*a62 + a31*a46*a52*a65 - a31*a46*a55*a62 - a32*a41*a55*a66 + a32*a41*a56*a65 + a32*a45*a51*a66 - a32*a45*a56*a61 - a32*a46*a51*a65 + a32*a46*a55*a61 + a35*a41*a52*a66 - a35*a41*a56*a62 - a35*a42*a51*a66 + a35*a42*a56*a61 + a35*a46*a51*a62 - a35*a46*a52*a61 - a36*a41*a52*a65 + a36*a41*a55*a62 + a36*a42*a51*a65 - a36*a42*a55*a61 - a36*a45*a51*a62 + a36*a45*a52*a61)*a24 + (a31*a44*a56*a65 - a31*a44*a55*a66 + a31*a45*a54*a66 - a31*a45*a56*a64 - a31*a46*a54*a65 + a31*a46*a55*a64 + a34*a41*a55*a66 - a34*a41*a56*a65 - a34*a45*a51*a66 + a34*a45*a56*a61 + a34*a46*a51*a65 - a34*a46*a55*a61 - a35*a41*a54*a66 + a35*a41*a56*a64 + a35*a44*a51*a66 - a35*a44*a56*a61 - a35*a46*a51*a64 + a35*a46*a54*a61 + a36*a41*a54*a65 - a36*a41*a55*a64 - a36*a44*a51*a65 + a36*a44*a55*a61 + a36*a45*a51*a64 - a36*a45*a54*a61)*a22 + (a32*a44*a55*a66 - a32*a44*a56*a65 - a32*a45*a54*a66 + a32*a45*a56*a64 + a32*a46*a54*a65 - a32*a46*a55*a64 - a34*a42*a55*a66 + a34*a42*a56*a65 + a34*a45*a52*a66 - a34*a45*a56*a62 - a34*a46*a52*a65 + a34*a46*a55*a62 + a35*a42*a54*a66 - a35*a42*a56*a64 - a35*a44*a52*a66 + a35*a44*a56*a62 + a35*a46*a52*a64 - a35*a46*a54*a62 - a36*a42*a54*a65 + a36*a42*a55*a64 + a36*a44*a52*a65 - a36*a44*a55*a62 - a36*a45*a52*a64 + a36*a45*a54*a62)*a21)*a13 
	+ ((a31*a43*a55*a64 - a31*a43*a54*a65 + a31*a44*a53*a65 - a31*a44*a55*a63 - a31*a45*a53*a64 + a31*a45*a54*a63 + a33*a41*a54*a65 - a33*a41*a55*a64 - a33*a44*a51*a65 + a33*a44*a55*a61 + a33*a45*a51*a64 - a33*a45*a54*a61 - a34*a41*a53*a65 + a34*a41*a55*a63 + a34*a43*a51*a65 - a34*a43*a55*a61 - a34*a45*a51*a63 + a34*a45*a53*a61 + a35*a41*a53*a64 - a35*a41*a54*a63 - a35*a43*a51*a64 + a35*a43*a54*a61 + a35*a44*a51*a63 - a35*a44*a53*a61)*a26 + (a31*a43*a54*a66 - a31*a43*a56*a64 - a31*a44*a53*a66 + a31*a44*a56*a63 + a31*a46*a53*a64 - a31*a46*a54*a63 - a33*a41*a54*a66 + a33*a41*a56*a64 + a33*a44*a51*a66 - a33*a44*a56*a61 - a33*a46*a51*a64 + a33*a46*a54*a61 + a34*a41*a53*a66 - a34*a41*a56*a63 - a34*a43*a51*a66 + a34*a43*a56*a61 + a34*a46*a51*a63 - a34*a46*a53*a61 - a36*a41*a53*a64 + a36*a41*a54*a63 + a36*a43*a51*a64 - a36*a43*a54*a61 - a36*a44*a51*a63 + a36*a44*a53*a61)*a25 + (a31*a43*a56*a65 - a31*a43*a55*a66 + a31*a45*a53*a66 - a31*a45*a56*a63 - a31*a46*a53*a65 + a31*a46*a55*a63 + a33*a41*a55*a66 - a33*a41*a56*a65 - a33*a45*a51*a66 + a33*a45*a56*a61 + a33*a46*a51*a65 - a33*a46*a55*a61 - a35*a41*a53*a66 + a35*a41*a56*a63 + a35*a43*a51*a66 - a35*a43*a56*a61 - a35*a46*a51*a63 + a35*a46*a53*a61 + a36*a41*a53*a65 - a36*a41*a55*a63 - a36*a43*a51*a65 + a36*a43*a55*a61 + a36*a45*a51*a63 - a36*a45*a53*a61)*a24 + (a31*a44*a55*a66 - a31*a44*a56*a65 - a31*a45*a54*a66 + a31*a45*a56*a64 + a31*a46*a54*a65 - a31*a46*a55*a64 - a34*a41*a55*a66 + a34*a41*a56*a65 + a34*a45*a51*a66 - a34*a45*a56*a61 - a34*a46*a51*a65 + a34*a46*a55*a61 + a35*a41*a54*a66 - a35*a41*a56*a64 - a35*a44*a51*a66 + a35*a44*a56*a61 + a35*a46*a51*a64 - a35*a46*a54*a61 - a36*a41*a54*a65 + a36*a41*a55*a64 + a36*a44*a51*a65 - a36*a44*a55*a61 - a36*a45*a51*a64 + a36*a45*a54*a61)*a23 + (a33*a44*a56*a65 - a33*a44*a55*a66 + a33*a45*a54*a66 - a33*a45*a56*a64 - a33*a46*a54*a65 + a33*a46*a55*a64 + a34*a43*a55*a66 - a34*a43*a56*a65 - a34*a45*a53*a66 + a34*a45*a56*a63 + a34*a46*a53*a65 - a34*a46*a55*a63 - a35*a43*a54*a66 + a35*a43*a56*a64 + a35*a44*a53*a66 - a35*a44*a56*a63 - a35*a46*a53*a64 + a35*a46*a54*a63 + a36*a43*a54*a65 - a36*a43*a55*a64 - a36*a44*a53*a65 + a36*a44*a55*a63 + a36*a45*a53*a64 - a36*a45*a54*a63)*a21)*a12 
	+ ((a32*a43*a54*a65 - a32*a43*a55*a64 - a32*a44*a53*a65 + a32*a44*a55*a63 + a32*a45*a53*a64 - a32*a45*a54*a63 - a33*a42*a54*a65 + a33*a42*a55*a64 + a33*a44*a52*a65 - a33*a44*a55*a62 - a33*a45*a52*a64 + a33*a45*a54*a62 + a34*a42*a53*a65 - a34*a42*a55*a63 - a34*a43*a52*a65 + a34*a43*a55*a62 + a34*a45*a52*a63 - a34*a45*a53*a62 - a35*a42*a53*a64 + a35*a42*a54*a63 + a35*a43*a52*a64 - a35*a43*a54*a62 - a35*a44*a52*a63 + a35*a44*a53*a62)*a26 + (a32*a43*a56*a64 - a32*a43*a54*a66 + a32*a44*a53*a66 - a32*a44*a56*a63 - a32*a46*a53*a64 + a32*a46*a54*a63 + a33*a42*a54*a66 - a33*a42*a56*a64 - a33*a44*a52*a66 + a33*a44*a56*a62 + a33*a46*a52*a64 - a33*a46*a54*a62 - a34*a42*a53*a66 + a34*a42*a56*a63 + a34*a43*a52*a66 - a34*a43*a56*a62 - a34*a46*a52*a63 + a34*a46*a53*a62 + a36*a42*a53*a64 - a36*a42*a54*a63 - a36*a43*a52*a64 + a36*a43*a54*a62 + a36*a44*a52*a63 - a36*a44*a53*a62)*a25 + (a32*a43*a55*a66 - a32*a43*a56*a65 - a32*a45*a53*a66 + a32*a45*a56*a63 + a32*a46*a53*a65 - a32*a46*a55*a63 - a33*a42*a55*a66 + a33*a42*a56*a65 + a33*a45*a52*a66 - a33*a45*a56*a62 - a33*a46*a52*a65 + a33*a46*a55*a62 + a35*a42*a53*a66 - a35*a42*a56*a63 - a35*a43*a52*a66 + a35*a43*a56*a62 + a35*a46*a52*a63 - a35*a46*a53*a62 - a36*a42*a53*a65 + a36*a42*a55*a63 + a36*a43*a52*a65 - a36*a43*a55*a62 - a36*a45*a52*a63 + a36*a45*a53*a62)*a24 + (a32*a44*a56*a65 - a32*a44*a55*a66 + a32*a45*a54*a66 - a32*a45*a56*a64 - a32*a46*a54*a65 + a32*a46*a55*a64 + a34*a42*a55*a66 - a34*a42*a56*a65 - a34*a45*a52*a66 + a34*a45*a56*a62 + a34*a46*a52*a65 - a34*a46*a55*a62 - a35*a42*a54*a66 + a35*a42*a56*a64 + a35*a44*a52*a66 - a35*a44*a56*a62 - a35*a46*a52*a64 + a35*a46*a54*a62 + a36*a42*a54*a65 - a36*a42*a55*a64 - a36*a44*a52*a65 + a36*a44*a55*a62 + a36*a45*a52*a64 - a36*a45*a54*a62)*a23 + (a33*a44*a55*a66 - a33*a44*a56*a65 - a33*a45*a54*a66 + a33*a45*a56*a64 + a33*a46*a54*a65 - a33*a46*a55*a64 - a34*a43*a55*a66 + a34*a43*a56*a65 + a34*a45*a53*a66 - a34*a45*a56*a63 - a34*a46*a53*a65 + a34*a46*a55*a63 + a35*a43*a54*a66 - a35*a43*a56*a64 - a35*a44*a53*a66 + a35*a44*a56*a63 + a35*a46*a53*a64 - a35*a46*a54*a63 - a36*a43*a54*a65 + a36*a43*a55*a64 + a36*a44*a53*a65 - a36*a44*a55*a63 - a36*a45*a53*a64 + a36*a45*a54*a63)*a22)*a11;

END_FUNCTION

// ---- AgiMaths/MatrixLib/matAdd.TcPOU
// C = A + B;
FUNCTION matAdd : BOOL
VAR_IN_OUT CONSTANT
	matA :ARRAY[*,*] OF LREAL;
	matB :ARRAY[*,*] OF LREAL;
END_VAR

VAR_IN_OUT 
	matC :ARRAY[*,*] OF LREAL;
END_VAR

VAR
	m,n :DINT;
	i,j, k :DINT;
 
END_VAR

m:=UPPER_BOUND(matC,1);
n:= UPPER_BOUND(matC,2);
ASSERT(UPPER_BOUND(matA,1)=m);
ASSERT(UPPER_BOUND(matA,2)=n);
ASSERT(UPPER_BOUND(matB,1)=m);
ASSERT(UPPER_BOUND(matB,2)=n);

FOR i:=1 TO m DO
	FOR j:=1 TO n DO
		matC[i,j]:=matA[i,j] + matB[i,j];
	END_FOR
END_FOR

END_FUNCTION

// ---- AgiMaths/MatrixLib/matSelfSub.TcPOU
// A -=B
FUNCTION matSelfSub : BOOL
VAR_IN_OUT;
	matA :ARRAY[*,*] OF LREAL;
END_VAR

VAR_IN_OUT CONSTANT
	matB :ARRAY[*,*] OF LREAL;
END_VAR

VAR
	m,n :DINT;
	i,j, k :DINT;
 
END_VAR

m:=UPPER_BOUND(matA,1);
n:= UPPER_BOUND(matA,2);
ASSERT(UPPER_BOUND(matB,1)=m);
ASSERT(UPPER_BOUND(matB,2)=n);
FOR i:=1 TO m DO
	FOR j:=1 TO n DO
		matA[i,j]:=matA[i,j]-matB[i,j];
	END_FOR
END_FOR

END_FUNCTION

// ---- AgiMaths/MatrixLib/vecSelfSub.TcPOU
// A -=B
FUNCTION vecSelfSub : BOOL
VAR_IN_OUT
	vecA :ARRAY[*] OF LREAL;
END_VAR

VAR_IN_OUT CONSTANT
	vecB :ARRAY[*] OF LREAL;
END_VAR

VAR
	m,i :DINT;
 
END_VAR

m:=UPPER_BOUND(vecA,1);
ASSERT(UPPER_BOUND(VecB,1)=m);

FOR i:=1 TO m DO
		vecA[i]:=vecA[i]-vecB[i];
END_FOR

END_FUNCTION

// ---- FBs_Auxiliary/FB_RiseEdgeCheck.TcPOU
FUNCTION_BLOCK FB_RiseEdgeCheck
VAR
	// last value
	m_lastValue :BOOL:=false;
END_VAR

METHOD check : BOOL
VAR_INPUT
	input :BOOL;
END_VAR
IF NOT(m_lastValue) AND input THEN
	check := TRUE;
ELSE
	check :=FALSE;
END_IF

m_lastValue := input;
END_METHOD

METHOD reset : BOOL
m_lastValue := false;
END_METHOD

END_FUNCTION_BLOCK

// ---- FBs_Auxiliary/FB_TON.TcPOU
FUNCTION_BLOCK FB_TON
VAR_INPUT
	IN : BOOL;
	PT : TIME;
END_VAR
VAR_OUTPUT
	Q : BOOL;
	ET : TIME;
END_VAR
VAR
	runTime : TIME;
	ctrlTime : TIME := T#1MS;
	zeroTime : TIME := T#0MS;
END_VAR

Q := FALSE;
IF IN THEN
	runTime := runTime + ctrlTime;
	IF runTime >= PT THEN
		Q := TRUE;
		runTime := PT;
	END_IF
ELSE
	runTime := zeroTime;
END_IF

END_FUNCTION_BLOCK

// ---- SafetyCheck/FB_Writer.TcPOU
FUNCTION_BLOCK FB_Writer
VAR_INPUT
	bWrite		: BOOL;		(* Rising edge starts program execution*)
	sNetId		: T_AmsNetId := '';	(* TwinCAT system network address *)
	sFileName	: T_MaxString;		(*  := 'HardDisk\TextModeGen.csv' CSV destination file path and name*) 
	pBuffer		: POINTER TO T_Buffer;
	Index		:UDINT;
END_VAR
VAR_OUTPUT
	bBusy: BOOL; 
	bError			: BOOL;
	nErrId			: UDINT;
END_VAR
VAR  
	fbFileOpen	: FB_FileOpen;(* Opens file *)
	fbFileClose	: FB_FileClose;(* Closes file *)
	fbAdsRdWrt	: FW_AdsRdWrt := ( nPort := AMSPORT_R3_SYSSERV, nIdxGrp := SYSTEMSERVICE_FPUTS, cbReadLen := 0, pReadBuff := 0 );	(* Writes one record (line) *)

 	_hFile			: UINT		:= 0;(* File handle of the source file *)
	_iStep			: DWORD 	:= 0;

	_iLen1: UDINT;
	_iLen2: UDINT;
	
	_iRow: UDINT;
	_iLastRow: UDINT;
	
	_iCol: UDINT;
	_iLastCol: UDINT;
	
	_iOffset: UDINT;
	
	_iCpy: UDINT;
	_pBuffer: PVOID;
	FristWriteFlag:BOOL;
	_sBuffer: STRING(MAX_BEFFER_SIZE);
END_VAR
 
VAR CONSTANT
	cs_Seperator: STRING[1]:= ';'; (*CSV字段分隔符*)
	cs_CarriageReturn: STRING[2]:= '$N'; (*换行符*)
	
	MAX_BEFFER_SIZE:UINT := 8192;(*每条ADS写命令写下去的内存大小*)
END_VAR

CASE _iStep OF
	0:	(* Wait for rising edge at bWrite variable *)
		IF bWrite THEN
			bWrite 		:= FALSE;
			bBusy 		:= TRUE;
			bError		:= FALSE;
			nErrId		:= 0;
			_hFile		:= 0; 
			_iStep 		:= 1;
			_iLastRow 	:= 0;
			_iLastCol   := 0;
		END_IF

	1:	(* Open source file *)
		fbFileOpen(  bExecute := FALSE  );
		fbFileOpen( 	sNetId := sNetId, sPathName := sFileName, nMode := FOPEN_MODEWRITE OR FOPEN_MODETEXT,(* Open file in TEXT mode! *)
						ePath := PATH_GENERIC, bExecute := TRUE );
		_iStep := 2;

	2:(* Wait until open not busy *)
		fbFileOpen( bExecute := FALSE, bError => bError, nErrID => nErrID, hFile => _hFile );
		IF NOT fbFileOpen.bBusy THEN
			IF NOT fbFileOpen.bError THEN
				_iStep := 3;
			ELSE(* Error: file not found? *)
				_iStep := 100;
			END_IF
		END_IF

	3:(* Convert one PLC record to CSV format *) 
		MEMSET(ADR(_sBuffer),0,MAX_BEFFER_SIZE);
		_iOffset := 0;
		_iCpy := 0;
		_pBuffer := ADR(_sBuffer);
		FOR _iRow := _iLastRow TO MAX_CSV_ROWS BY 1 DO
			FOR _iCol := _iLastCol TO MAX_CSV_COLUMNS BY 1 DO 
				_iLen1 := LEN(pBuffer^[  _iRow][_iCol]);
				_iLen2 := LEN(cs_Seperator); 
				IF (_iOffset + _iLen1 + _iLen2 + 1) < MAX_BEFFER_SIZE THEN 
					_iCpy := FW_MemCpy(_pBuffer + _iOffset, ADR(pBuffer^[  _iRow][_iCol]), _iLen1);
					_iOffset := _iOffset + _iCpy;
					IF  _iCol < MAX_CSV_COLUMNS THEN
						_iCpy := FW_MemCpy(_pBuffer + _iOffset, ADR(cs_Seperator), _iLen2);
						_iOffset := _iOffset + _iCpy;
					END_IF
				ELSE
					_iLastRow := _iRow;
					_iLastCol := _iCol;
					_iStep := 4;(* Write record to the file *)
					RETURN;	
				END_IF
			END_FOR 
			_iLen2 := LEN(cs_CarriageReturn); 
			_iCpy:= FW_MemCpy(_pBuffer + _iOffset, ADR(cs_CarriageReturn), _iLen2);
			_iOffset := _iOffset + _iCpy;
			_iLastCol := 0;
		END_FOR 
		_iStep := 4;(* Write record to the file *) 
	4:	(* Write single text line *) 
		fbAdsRdWrt( bExecute := FALSE ); 
		fbAdsRdWrt( sNetId := sNetId, nIdxOffs := _hFile, cbWriteLen := _iOffset + 1(*inclusive terminating NULL*), pWriteBuff := ADR(_sBuffer),
			bExecute := TRUE, tTimeout := DEFAULT_ADS_TIMEOUT, bBusy=>bBusy, bError=>bError, nErrID=>nErrID );
		_iStep := 5;

	5:(* Wait until write not busy *)
		fbAdsRdWrt( bExecute := FALSE, bError => bError, nErrID => nErrID );
		IF NOT fbAdsRdWrt.bBusy THEN
			IF NOT fbAdsRdWrt.bError THEN 
				_iStep := 3;(* Write next record *)
				IF _iRow >= MAX_CSV_ROWS THEN
					_iStep := 10;
				END_IF
			ELSE(* Error *)
				_iStep := 100;
			END_IF
		END_IF

	10:	(* Close source file *)
		fbFileClose( bExecute := FALSE );
		fbFileClose( sNetId := sNetId, hFile := _hFile, bExecute := TRUE );
		_iStep := 11;

	11:(* Wait until close not busy *)
		fbFileClose( bExecute := FALSE, bError => bError, nErrID => nErrID );
		IF ( NOT fbFileClose.bBusy ) THEN
			_hFile := 0;
			_iStep := 100;
		END_IF

	100: (* Error or ready step => cleanup *)
		IF ( _hFile <> 0 ) THEN
			_iStep := 10; (* Close the source file *)
		ELSE
			bBusy := FALSE;
			_iStep := 0;	(* Ready *) 
		END_IF

END_CASE

END_FUNCTION_BLOCK

// ---- Sandbox/FB_CartCheck.TcPOU
FUNCTION_BLOCK FB_CartCheck
VAR_INPUT
END_VAR
VAR_OUTPUT
END_VAR
VAR
	// joint error flag
	m_jointErrFlag :ARRAY[1..4] OF BOOL:=[4(FALSE)];
	
	// joint control error flag
	m_jntCtrlErrFlag :vec4b;
	m_jntCtrlErrCounts :Vec4i;
	m_jntEncErr :Vec4d;
	
	// joint encoder error flag
	m_jntEncErrFlag :vec4b;
	m_jntEncErrCounts :Vec4i;
	m_jntCtrlErr : Vec4d;
	
	// joint velocity error flag
	m_jntVelErrFlag :vec4b;
	m_jntVelErrCounts  :Vec4i;
	
	// joint position limit error flag
	m_jntLimitErrFlag :Vec4b;
	m_jntLimitErrCounts :Vec4i;
	
END_VAR

METHOD check : BOOL
VAR_IN_OUT CONSTANT
	i_cartStatus : ST_CartStatus;
	i_cartJointData :ST_CartJointData;
END_VAR
VAR_OUTPUT
	o_errorFlag :ARRAY[1..4] OF BOOL ;
END_VAR

VAR
	i ,j:INT ;
END_VAR
// return if cart not init
IF NOT(i_cartStatus.m_initFlag) THEN
	RETURN;
END_IF

// joint control error
jntCtrlErrCheck(i_cartJointData.m_cmdJntPos, i_cartJointData.m_curJntPos);

// encoder error
jntEncErrCheck(i_cartJointData.m_curMotorPos, i_cartJointData.m_curLinkPos);

// joint velocity error
jntVelCheck(i_cartJointData.m_curJntVel);

// joint limit 
jntLimitCheck(i_cartJointData.m_curJntPos);
	
FOR i:=1 TO 4 DO 
	// stop check if arm is already in error state
	IF  m_jointErrFlag[i] THEN 
		CONTINUE;
	END_IF
	
	// final arm error status check
	IF m_jntCtrlErrFlag[i] OR  m_jntEncErrFlag[i] OR m_jntVelErrFlag[i] OR m_jntLimitErrFlag[i] THEN
		m_jointErrFlag[i]:=TRUE;
		EXIT;
	END_IF
	
END_FOR

o_errorFlag:=m_jointErrFlag;
END_METHOD

METHOD jntCtrlErrCheck : BOOL
VAR_INput
	i_cmdJntPos : Vec4d;
	i_curJntPos : Vec4d;
END_VAR

VAR
	i :INT;
END_VAR
// joint error check
FOR i:=1 TO 4 DO 
	// stop check if arm is already in error state
	IF m_jointErrFlag[i] THEN 
		CONTINUE;
	END_IF
	
	// error
	m_jntCtrlErr[i]:= i_cmdJntPos[i]-i_curJntPos[i];
	
	//check
	IF  ABS(m_jntCtrlErr[i]) > g_cartMaxJntCtrlErr[i] THEN
		m_jntCtrlErrCounts[i]:=m_jntCtrlErrCounts[i]+1;
	ELSE
		m_jntCtrlErrCounts[i] :=0;	
	END_IF
	m_jntCtrlErrFlag[i]:= m_jntCtrlErrCounts[i]>=g_faultTriggerCounts;
END_FOR
END_METHOD

METHOD jntEncErrCheck : BOOL
VAR_INput
	i_motorJntPos : Vec4d;
	i_linkJntPos : Vec4d;
END_VAR


VAR
	i :INT;
END_VAR
// joint error check
FOR i:=1 TO 4 DO 
	// stop check if arm is already in error state
	IF  m_jointErrFlag[i] THEN 
		CONTINUE;
	END_IF
	
	// error
	m_jntEncErr[i]:=i_motorJntPos[i]-i_linkJntPos[i];
	
	// check
	IF  ABS(m_jntEncErr[i]) > g_cartMaxJntEncErr[i] THEN
		m_jntEncErrCounts[i]:=m_jntEncErrCounts[i]+1;
	ELSE
		m_jntEncErrCounts[i] :=0;
	END_IF
	m_jntEncErrFlag[i]:= m_jntEncErrCounts[i]>=g_faultTriggerCounts;
END_FOR
END_METHOD

METHOD jntLimitCheck : bool
VAR_INPUT
	i_curJntPos : Vec4d;
END_VAR

VAR
	i:INT;
END_VAR
// joint position limit check
FOR i:=1 TO 4 DO 
	// stop check if arm is already in error state
	IF m_jointErrFlag[i] THEN 
		CONTINUE;
	END_IF
	
	// check
	IF  i_curJntPos[i] > GVL_CartJointParameters.g_maxJntPos[i] + g_cartJntPosLimitBuffer[i] OR
		i_curJntPos[i] < GVL_CartJointParameters.g_minJntPos[i] - g_cartJntPosLimitBuffer[i] THEN
		m_jntLimitErrCounts[i]:=m_jntLimitErrCounts[i]+1;
	ELSE
		m_jntLimitErrCounts[i] :=0;	
	END_IF
	m_jntLimitErrFlag[i]:= m_jntLimitErrCounts[i]>=g_faultTriggerCounts;
END_FOR
END_METHOD

METHOD jntVelCheck : bool
VAR_INPUT
	i_curJntVel : Vec4d;
END_VAR

VAR
	i:INT;
END_VAR
// joint velocity check
FOR i:=1 TO 4 DO 
	// stop check if arm is already in error state
	IF m_jointErrFlag[i] THEN 
		CONTINUE;
	END_IF
	
	// check
	IF  ABS(i_curJntVel[i]) > g_cartMaxJntVel[i] THEN
		m_jntVelErrCounts[i]:=m_jntVelErrCounts[i]+1;
	ELSE
		m_jntVelErrCounts[i] :=0;
	END_IF
	m_jntVelErrFlag[i]:= m_jntVelErrCounts[i]>=g_faultTriggerCounts;
END_FOR
END_METHOD

END_FUNCTION_BLOCK

// ---- Sandbox/FB_MasterArmCheck.TcPOU
FUNCTION_BLOCK FB_MasterArmCheck
VAR_INPUT
END_VAR
VAR_OUTPUT
END_VAR
VAR
	// whole arm error flag
	m_armErrFlag :ARRAY[1..g_mArmNum] OF BOOL:=[2(FALSE)];
	
	// cartesian pose error flag
	m_cartPoseErrFlag :ARRAY[1..g_mArmNum] OF BOOL;
	m_cartPoseErrCounts:ARRAY[1..g_mArmNum] OF INT;
	m_cartPosErr :ARRAY[1..g_mArmNum] OF Vec3d;		// cartesian position error
	m_cartOriErr:ARRAY[1..g_mArmNum] OF  Vec3d;	// cartesian rotation angle (angle  * axis)
	
	// joint control error flag
	m_jntCtrlErrFlag :ARRAY[1..g_mArmNum] OF Vec7b;
	m_jntCtrlErrCounts :ARRAY[1..g_mArmNum] OF Vec7i;
	m_jntCtrlErr:ARRAY[1..g_mArmNum]  OF Vec7d;		// joint position control error
	
	// joint encoder error flag
	m_jntEncErrFlag :ARRAY[1..g_mArmNum] OF Vec7b;
	m_jntEncErrCounts :ARRAY[1..g_mArmNum] OF Vec7i ;
	m_jntEncErr:ARRAY[1..g_mArmNum]  OF Vec7d;		// motor and joint encoder error
	
	// joint velocity error flag
	m_jntVelErrFlag :ARRAY[1..g_mArmNum] OF Vec7b;
	m_jntVelErrCounts :ARRAY[1..g_mArmNum] OF Vec7i;
	
	// joint position limit error flag
	m_jntLimitErrFlag :ARRAY[1..g_mArmNum] OF Vec7b;
	m_jntLimitErrCounts :ARRAY[1..g_mArmNum] OF Vec7i;
	
END_VAR

METHOD check : BOOL
VAR_IN_OUT CONSTANT
	i_masterStatus : ST_MasterStatus;
	i_masterJointData :ST_MasterJointData;
END_VAR
VAR_OUTPUT
	o_errorFlag :ARRAY[1..g_mArmNum] OF BOOL ;
END_VAR

VAR
	i ,j:INT ;
END_VAR
// calculate error
FOR i:=1 TO g_mArmNum DO 
	// stop check if arm is already in error state
	IF m_armErrFlag[i] OR i_masterStatus.m_armState[i] = MasterArmState_Error THEN 
		CONTINUE;
	END_IF
	
	// NOT check cartesion pose error
	m_cartPoseErrFlag[i]:=FALSE;
	//m_cartPoseErrFlag[i]:=poseErrCheck(i_masterStatus.m_cmdArmPose[i],  i_masterStatus.m_curArmPose[i],
	//										m_cartPoseErrCounts[i], m_cartPosErr[i], m_cartOriErr[i]);
	
	// joint control error
	m_jntCtrlErrFlag[i]:=jntCtrlErrCheck(i_masterJointData.m_cmdJntPos[i], i_masterJointData.m_curJntPos[i],
										m_jntCtrlErrCounts[i], m_jntCtrlErr[i]);
	
	// encoder error
	m_jntEncErrFlag[i]:=jntEncErrCheck(i_masterJointData.m_curMotorPos[i], i_masterJointData.m_curLinkPos[i],
										m_jntEncErrCounts[i], m_jntEncErr[i]);
	
	// joint limit error
	m_jntLimitErrFlag[i]:=jntLimitErrCheck(i,i_masterJointData.m_curJntPos[i],m_jntLimitErrCounts[i]);
	IF i_masterStatus.m_armState[i] = MasterArmState_Init THEN
		m_jntLimitErrFlag[i][7] := false;
	END_IF
										
	// final arm error status check
	IF  m_cartPoseErrFlag[i] THEN
		m_armErrFlag[i]:=TRUE;
		CONTINUE;
	END_IF
	
	FOR j:=1 TO g_mJntNum DO 
		//IF m_jntCtrlErrFlag[i][j] OR m_jntEncErrFlag[i][j] OR m_jntVelErrFlag[i][j] OR m_jntLimitErrFlag[i][j] THEN
		IF m_jntEncErrFlag[i][j] OR m_jntVelErrFlag[i][j] OR m_jntLimitErrFlag[i][j] THEN
			m_armErrFlag[i]:=TRUE;
			EXIT;
		END_IF
	END_FOR
	
END_FOR

o_errorFlag:=m_armErrFlag;
END_METHOD

METHOD jntCtrlErrCheck : Vec7b
VAR_INput
	i_cmdJntPos : Vec7d;
	i_curJntPos : Vec7d;
END_VAR
VAR_IN_OUT
	r_errCount:Vec7i;
	r_jntCtrlErr :Vec7d;
END_VAR

VAR
	i :INT;
	err:Vec7d;
END_VAR
vecSub(i_cmdJntPos,i_curJntPos,  err);
r_jntCtrlErr:=err;

// joint error check
FOR i:=1 TO g_mJntNum DO 
	IF  ABS(r_jntCtrlErr[i]) > g_maxJntCtrlErr THEN
		r_errCount[i]:=r_errCount[i]+1;
	ELSE
		r_errCount[i] :=0;	
	END_IF
	jntCtrlErrCheck[i]:= r_errCount[i]>=g_faultTriggerCounts;
END_FOR
END_METHOD

METHOD jntEncErrCheck : Vec7b
VAR_INput
	i_motorJntPos : Vec7d;
	i_linkJntPos : Vec7d;
END_VAR
VAR_IN_OUT
	r_errCount:Vec7i;
	r_jntEncErr :Vec7d;
END_VAR

VAR
	i :INT;
	err:Vec7d;
END_VAR
vecSub(i_motorJntPos,i_linkJntPos,  err);
r_jntEncErr:=err;

// joint error check
FOR i:=1 TO g_mJntNum DO 
	IF  ABS(r_jntEncErr[i]) > g_maxJntEncErr THEN
		r_errCount[i]:=r_errCount[i]+1;
	ELSE
		r_errCount[i] :=0;
	END_IF
	jntEncErrCheck[i]:= r_errCount[i]>=g_faultTriggerCounts;
END_FOR
END_METHOD

METHOD jntLimitErrCheck : Vec7b
VAR_INPUT
	i_armIdx:INT;
	i_curJntPos : Vec7d;
END_VAR
VAR_IN_OUT
	r_errCount:Vec7i;
END_VAR

VAR
	i :INT;
END_VAR
i_curJntPos[4]:=i_curJntPos[4]+i_curJntPos[3]-i_curJntPos[2]-pi/2;//q4DH=q4motor+q8-q2-90;  

// joint limit check
FOR i:=1 TO 7 DO 
	IF  i_curJntPos[i] > GVL_ArmJointParameters.g_maxJntPos[i_armIdx,i] + g_armJntPosLimitBuffer[i] OR
		i_curJntPos[i] < GVL_ArmJointParameters.g_minJntPos[i_armIdx,i] - g_armJntPosLimitBuffer[i] THEN
		r_errCount[i]:=r_errCount[i]+1;
	ELSE
		r_errCount[i] :=0;	
	END_IF
	jntLimitErrCheck[i]:= r_errCount[i]>=g_faultTriggerCounts;
END_FOR
END_METHOD

METHOD poseErrCheck : BOOL
VAR_INPUT
	i_cmdPose : ST_Frame;
	i_curPose :ST_Frame;
END_VAR
VAR_IN_OUT
	r_errCount:INT;
	r_posErr :Vec3d;
	r_oriErr :Vec3d;
END_VAR

VAR
	posErr,oriErr:Vec3d;
	matT,rotErr:Mat3d;
	errAngle :LREAL;
	errAxis :Vec3d;
END_VAR

vecSub(i_cmdPose.m_pos, i_curPose.m_pos,posErr);
r_posErr:=posErr;

matTranspose(i_cmdPose.m_rot, matT);
matMultiply(matT,i_curPose.m_rot, rotErr);
rot2AngAxis(rotErr, angle=>errAngle, axis=>errAxis);
vecMultiNum(errAxis, errAngle,oriErr);
r_oriErr:=oriErr;
	
IF  norm(posErr)>g_maxCartPosErr OR norm(oriErr)> g_maxCartOriErr THEN
	r_errCount:= r_errCount +1;
ELSE 
	r_errCount:=0;
END_IF
poseErrCheck:= r_errCount >= g_faultTriggerCounts;
END_METHOD

END_FUNCTION_BLOCK

// ---- Sandbox/FB_RedunJntControl_bak2.TcPOU
// Author: Feijian Ni
// Date: 2023.11.22
FUNCTION_BLOCK FB_RedunJntControl_bak2
VAR_INPUT
END_VAR
VAR_OUTPUT
END_VAR
VAR
	// static velocity threshold
	m_staticVelThres :LREAL := 90 *g_deg2Rad;
	
	// static threshold of joint bias
	m_staticBiasThres :LREAL := 35 *g_deg2Rad;
	
	// rudundancy track flag
	m_trackFlag :BOOL;
	
	// joint4 track tolerance
	m_joint4TrackTol :LREAL :=1*g_deg2rad;
	
	// current manipulation velocity
	m_curManipWVel :LREAL :=0;
	
	// joint4 limit buffer
	m_jntLimitBuffer : LREAL :=2.5*g_deg2Rad;
	
	// control paramters for redundant joint4 position control
(*	m_redunJntKp: LREAL:=8.0;
	m_redunJntKd:LREAL:=0.2;
	m_redunJntKi:LREAL:=100; *)
	m_redunJntKp: LREAL:=3.0;
	m_redunJntKd:LREAL:=0.1;
	m_redunJntKi:LREAL:=0;
	m_redunJntKiLimit: LREAL:=200;
	m_redunJntCtrlLimit:LREAL:=1000;

	// max vel and acc for joint4 motion
	m_jnt4MaxFollowVel :LREAL :=2*pi;
	m_jnt4MaxFollowAcc :LREAL :=6*pi;
	m_jnt4MinFollowAcc :LREAL :=2*pi;
	m_jnt4MinAccVel:LREAL:= 60 *g_deg2Rad;
	m_jnt4MaxAccVel:LREAL:= 150 *g_deg2Rad;

	// final target position of joint4 in motor (not DH , same for below defination) 
	m_jnt4TargetPos: LREAL;
	
	// OTG for joint4 motion
	m_trajFilter :FB_secOrdTrajFilter;
	
	// command joint4 position and veloicty in motor for next cycle
	m_cmdJntPos: LREAL;
	m_cmdJntVel: LREAL;
	m_cmdJntAcc: LREAL;

	// PID for joint position
	m_jntPIDCtrl: FB_PID;
	m_jntCtrlTrq: LREAL;
	
END_VAR

METHOD PROTECTED calcRedunPos : BOOL
VAR_IN_OUT CONSTANT
	i_masterArm :FB_MasterArm;
END_VAR

VAR 
	j6Bias,j5Bias :LREAL;
	curJntPos : Vec7d;
	jnt4LinkPos, jnt4TargetLinkPos :LREAL;
END_VAR
// compute desired joint4 link position
curJntPos :=  i_masterArm.curLinkPos;
jnt4LinkPos:=i_masterArm.jnt4MotorToLink(curJntPos[2],curJntPos[3],curJntPos[4]);
IF 1= i_masterArm.armIdx THEN
	j6Bias :=curJntPos[6]+PI/2;
ELSE 
	j6Bias := curJntPos[6]-PI/2;
END_IF

// scale track motion near redundant singularity
j5Bias :=  LIMIT (0, ABS(curJntPos[5] -pi), pi/2);
j6Bias := j6Bias * ABS(COS(j5Bias));
jnt4TargetLinkPos := LIMIT(GVL_ArmJointParameters.g_minJntPos[i_masterArm.armIdx,4]+m_jntLimitBuffer, 
			jnt4LinkPos-j6Bias,GVL_ArmJointParameters.g_maxJntPos[i_masterArm.armIdx,4]-m_jntLimitBuffer); 
			
// convert from link position to motor position
m_jnt4TargetPos:=i_masterArm.jnt4LinkToMotor(curJntPos[2], curJntPos[3], jnt4TargetLinkPos);
END_METHOD

METHOD init : BOOL
VAR_IN_OUT CONSTANT
	i_masterArm :FB_MasterArm;
END_VAR
VAR
	currentRatioMotor2Jnt:LREAL;
END_VAR
m_cmdJntPos:=i_masterArm.curJntPos[4];
m_jnt4TargetPos:=m_cmdJntPos;
m_cmdJntVel:=0;

// init controller
currentRatioMotor2Jnt:=GVL_ArmJointParameters.g_motorTrqConst[4]*GVL_ArmJointParameters.g_motorReduction[4]/1000;
m_jntPIDCtrl.init(g_armCtrlCycleTime,m_redunJntKp,m_redunJntKd,m_redunJntKi,
		m_redunJntKiLimit* currentRatioMotor2Jnt,	m_redunJntCtrlLimit*currentRatioMotor2Jnt);

// init OTG
m_trajFilter.init(m_cmdJntPos,m_cmdJntVel,m_jnt4MaxFollowVel,m_jnt4MaxFollowAcc,g_armCtrlCycleTime);
END_METHOD

METHOD run : LREAL
VAR_IN_OUT CONSTANT
	i_masterArm :FB_MasterArm;
END_VAR
VAR_INPUT
	i_followEnable :BOOL;
END_VAR


VAR
	maxAcc, minDec:LREAL;
END_VAR
// check if arm is static
m_trackFlag := startTrack(i_masterArm);
	
// determin target position of joint4
IF i_followEnable THEN
	// update target redundant joint position
	IF  m_trackFlag THEN
		calcRedunPos(i_masterArm);
	ELSE
		// no control in static state
		IF ABS(m_cmdJntPos-m_jnt4TargetPos)< m_joint4TrackTol THEN
			m_jnt4TargetPos := i_masterArm.curJntPos[4];
			m_cmdJntPos :=i_masterArm.curJntPos[4];
			m_cmdJntVel:=0;
			m_jntPIDCtrl.reset();
			m_trajFilter.init(m_cmdJntPos,m_cmdJntVel,m_jnt4MaxFollowVel,m_jnt4MaxFollowAcc,g_armCtrlCycleTime);
		END_IF
	END_IF
END_IF

	
// scale following acceleration based on yaw velocity
maxAcc:=(m_jnt4MaxFollowAcc-m_jnt4MinFollowAcc)*(ABS(i_masterArm.curCartTwist[6])-m_jnt4MinAccVel)/(m_jnt4MaxAccVel-m_jnt4MinAccVel)+m_jnt4MinFollowAcc;
maxAcc := LIMIT(m_jnt4MinFollowAcc,maxAcc, m_jnt4MaxFollowAcc);
minDec:=m_trajFilter.minDec(m_jnt4TargetPos);
maxAcc := MAX(maxAcc, minDec);

// run OTG
m_trajFilter.maxV:=m_curManipWVel;
m_trajFilter.maxA:=maxAcc;
m_trajFilter.run(m_jnt4TargetPos, 0.0, o_cmdAcc=>m_cmdJntAcc,o_cmdVel=>m_cmdJntVel, o_cmdPos=>m_cmdJntPos);

// joint position control torque control
m_jntCtrlTrq:=m_jntPIDCtrl.run(m_cmdJntPos,i_masterArm.curJntPos[4], m_cmdJntVel, i_masterArm.curJntVel[4]);
//m_jntCtrlTrq:= m_jntCtrlTrq+i_masterArm.massMat[4,4]*m_cmdJntAcc;

run:=m_jntCtrlTrq;
END_METHOD

METHOD startTrack : BOOL
VAR_IN_OUT CONSTANT
	i_masterArm :FB_MasterArm;
END_VAR
VAR
	j6Bias :LREAL;
	curJntPos : Vec7d;
	wVelWrd, wVelLocal :Vec3d;
	rotT:Mat3d;
END_VAR
curJntPos :=  i_masterArm.curLinkPos;
IF 1= i_masterArm.armIdx THEN
	j6Bias :=curJntPos[6]+PI/2;
ELSE 
	j6Bias := curJntPos[6]-PI/2;
END_IF

wVelWrd[1]:= i_masterArm.m_curCartLinkTwist[4];
wVelWrd[2]:= i_masterArm.m_curCartLinkTwist[5];
wVelWrd[3]:= i_masterArm.m_curCartLinkTwist[6];

matTranspose(i_masterArm.curCartPose.m_rot, rotT);
matMultiVec(rotT, wVelWrd, wVelLocal);

wVelLocal[3]:=0;
m_curManipWVel:=norm(wVelLocal);

IF (m_curManipWVel> m_staticVelThres AND i_masterArm.m_curLinkVel[6] * j6Bias > 0)  OR ABS(j6Bias)> m_staticBiasThres THEN
	startTrack := TRUE;
ELSE
	startTrack :=FALSE;
END_IF
END_METHOD

END_FUNCTION_BLOCK

// ---- Sandbox/FB_RedunJntControl_bak.TcPOU
// Author: Feijian Ni
// Date: 2023.11.22
FUNCTION_BLOCK FB_RedunJntControl_bak
VAR_INPUT
END_VAR
VAR_OUTPUT
END_VAR
VAR
	// joint4 backlash
	m_joint4Backlash :LREAL :=10*g_deg2rad;
	
	// control paramters for redundant joint4 position control
(*	m_redunJntKp: LREAL:=8.0;
	m_redunJntKd:LREAL:=0.2;
	m_redunJntKi:LREAL:=100; *)
	m_redunJntKp: LREAL:=3.0;
	m_redunJntKd:LREAL:=0.1;
	m_redunJntKi:LREAL:=10;
	m_redunJntKiLimit: LREAL:=200;
	m_redunJntCtrlLimit:LREAL:=1000;
	
	m_jntLimitBuffer : LREAL :=5.0*g_deg2Rad;
	
	// arm static variables
	m_staticVelThres :LREAL := 5.0 *g_deg2Rad;
	m_staticTimeThres :LREAL :=0.2;
	m_staticTime :LREAL;
	m_staticFlag :BOOL;
		
	// max vel and acc for joint4 motion
	m_jnt4MaxFollowVel :LREAL :=2*pi;
	m_jnt4MaxFollowAcc :LREAL :=6*pi;
	m_jnt4MinFollowAcc :LREAL :=3*pi;
	m_jnt4MinAccVel:LREAL:= 0.5*pi;
	m_jnt4MaxAccVel:LREAL:= 1.0*pi;

	// final target position of joint4 in motor (not DH , same for below defination) 
	m_jnt4TargetPos: LREAL;
	
	// OTG for joint4 motion
	m_trajFilter :FB_secOrdTrajFilter;
	
	// command joint4 position and veloicty in motor for next cycle
	m_cmdJntPos: LREAL;
	m_cmdJntVel: LREAL;
	m_cmdJntAcc: LREAL;

	// PID for joint position
	m_jntPIDCtrl: FB_PID;
	m_jntCtrlTrq: LREAL;

	
END_VAR

METHOD PROTECTED calcRedunPos : BOOL
VAR_IN_OUT CONSTANT
	i_masterArm :FB_MasterArm;
END_VAR

VAR 
	j6Bias,j5Bias :LREAL;
	curJntPos : Vec7d;
	jnt4LinkPos, jnt4TargetLinkPos :LREAL;
END_VAR
// compute desired joint4 link position
curJntPos :=  i_masterArm.curLinkPos;
jnt4LinkPos:=i_masterArm.jnt4MotorToLink(curJntPos[2],curJntPos[3],curJntPos[4]);
IF 1= i_masterArm.armIdx THEN
	j6Bias :=curJntPos[6]+PI/2;
ELSE 
	j6Bias := curJntPos[6]-PI/2;
END_IF

// scale track motion near redundant singularity
j5Bias :=  LIMIT (0, ABS(curJntPos[5] -pi), pi/2);
j6Bias := j6Bias * ABS(COS(j5Bias));
jnt4TargetLinkPos := LIMIT(GVL_ArmJointParameters.g_minJntPos[i_masterArm.armIdx,4]+m_jntLimitBuffer, 
			jnt4LinkPos-j6Bias,GVL_ArmJointParameters.g_maxJntPos[i_masterArm.armIdx,4]-m_jntLimitBuffer); 
			
// convert from link position to motor position
m_jnt4TargetPos:=i_masterArm.jnt4LinkToMotor(curJntPos[2], curJntPos[3], jnt4TargetLinkPos);
END_METHOD

METHOD init : BOOL
VAR_IN_OUT CONSTANT
	i_masterArm :FB_MasterArm;
END_VAR
VAR
	currentRatioMotor2Jnt:LREAL;
END_VAR
m_cmdJntPos:=i_masterArm.curJntPos[4];
m_jnt4TargetPos:=m_cmdJntPos;
m_cmdJntVel:=0;

// init controller
currentRatioMotor2Jnt:=GVL_ArmJointParameters.g_motorTrqConst[4]*GVL_ArmJointParameters.g_motorReduction[4]/1000;
m_jntPIDCtrl.init(g_armCtrlCycleTime,m_redunJntKp,m_redunJntKd,m_redunJntKi,
		m_redunJntKiLimit* currentRatioMotor2Jnt,	m_redunJntCtrlLimit*currentRatioMotor2Jnt);

// init OTG
m_trajFilter.init(m_cmdJntPos,m_cmdJntVel,m_jnt4MaxFollowVel,m_jnt4MinFollowAcc,g_armCtrlCycleTime);
END_METHOD

METHOD isStatic : BOOL
VAR_IN_OUT CONSTANT
	i_masterArm :FB_MasterArm;
END_VAR
VAR
	wVelWrd, wVelLocal :Vec3d;
	rotT :Mat3d;
END_VAR
wVelWrd[1]:=i_masterArm.curCartTwist[4];
wVelWrd[2]:=i_masterArm.curCartTwist[5];
wVelWrd[3]:=i_masterArm.curCartTwist[6];
matTranspose(i_masterArm.curCartPose.m_rot, rotT);
matMultiVec(rotT, wVelWrd, wVelLocal);
wVelLocal[3]:=0;

IF norm(wVelLocal) <m_staticVelThres THEN
	m_staticTime := m_staticTime + g_armCtrlCycleTime;
ELSE
	m_staticTime :=0;
END_IF

isStatic := m_staticTime >= m_staticTimeThres;
END_METHOD

METHOD run : LREAL
VAR_IN_OUT CONSTANT
	i_masterArm :FB_MasterArm;
END_VAR
VAR_INPUT
	i_followEnable :BOOL;
END_VAR


VAR
	maxAcc, minDec:LREAL;
END_VAR
// check if arm is static
m_staticFlag := isStatic(i_masterArm);
	
// determin target position of joint4
IF i_followEnable THEN
	// no control in static state
	IF  m_staticFlag THEN
		m_jnt4TargetPos := i_masterArm.curJntPos[4];
		m_cmdJntPos :=i_masterArm.curJntPos[4];
		m_cmdJntVel:=0;
		m_jntPIDCtrl.reset();
		m_trajFilter.init(m_cmdJntPos,m_cmdJntVel,m_jnt4MaxFollowVel,m_jnt4MinFollowAcc,g_armCtrlCycleTime);
	// update target redundant joint position
	ELSE
		calcRedunPos(i_masterArm);
	END_IF
END_IF
	
// scale following acceleration based on yaw velocity
maxAcc:=(m_jnt4MaxFollowAcc-m_jnt4MinFollowAcc)*(ABS(i_masterArm.curCartTwist[6])-m_jnt4MinAccVel)/(m_jnt4MaxAccVel-m_jnt4MinAccVel)+m_jnt4MinFollowAcc;
maxAcc := LIMIT(m_jnt4MinFollowAcc,maxAcc, m_jnt4MaxFollowAcc);
minDec:=m_trajFilter.minDec(m_jnt4TargetPos);
maxAcc := MAX(maxAcc, minDec);

// run OTG
m_trajFilter.maxA:=maxAcc;
m_trajFilter.run(m_jnt4TargetPos, 0.0, o_cmdAcc=>m_cmdJntAcc,o_cmdVel=>m_cmdJntVel, o_cmdPos=>m_cmdJntPos);

// joint position control torque control
m_jntCtrlTrq:=m_jntPIDCtrl.run(m_cmdJntPos,i_masterArm.curJntPos[4], m_cmdJntVel, i_masterArm.curJntVel[4]);
//m_jntCtrlTrq:= m_jntCtrlTrq+i_masterArm.massMat[4,4]*m_cmdJntAcc;

run:=m_jntCtrlTrq;
END_METHOD

END_FUNCTION_BLOCK
